(* CODESYS project Proje_1.project
   Title: Step
   Version: 0.0.0.0
   Author: MustafaZahid

Project tree, tasks and I/O mapping:
  MyController : TM241C24T/U, Schneider Electric, order no. TM241C24T/U, version 4.0.6.18
    application Application
      task MAST (cyclic, interval 20 ms, priority 15, watchdog 100 ms x 1) calls POU
      global variables GVL
      program POU [LD]
      FunctionBlocks/
        function block Motor_Administration [LD]
        function block Axis_Limits [LD]
    DI : Digital Inputs, Schneider Electric, version 4.0.6.18
        input  iwDI_IW0 : WORD  // IW0
        input  Application.POU.Sensor_1 : BOOL  // IW0.I0
        input  ibDI_IB1 : BYTE  // IB1
    DQ : Digital Outputs, Schneider Electric, version 4.0.6.18
        settings: Outputs Usage = 3
        output qwDQ_QW0 : WORD  // QW0
        output qbDQ_QB1 : BYTE  // QB1
    Counters : Counters, Schneider Electric, version 4.0.6.18
    Pulse_Generators : Pulse Generators, Schneider Electric, version 4.0.6.18
        settings: Instance name = 'Axis_1'; PROBE input History = 'old=0 new=-1'; REF input History = 'old=0 new=-1'; B output History = 'old=-1 new=1'; A output History = 'old=-1 new=0'; Temporary Instance name = 'Axis_1'
    Cartridge_1 : Cartridge, Schneider Electric, version 4.0.6.18
    IO_Bus : IO bus - TM3, Schneider Electric, version 4.0.6.18
    COM_Bus : COM bus, Schneider Electric, version 4.0.6.18
    Serial_Line_1 : Serial line, Schneider Electric, version 4.0.6.18
      SoMachine_Network_Manager : SoMachine-Network Manager, Schneider Electric, version 4.0.0.2
    Serial_Line_2 : Serial line, Schneider Electric, version 4.0.6.18
      Modbus_Manager : Modbus Manager, Schneider Electric, version 4.0.0.2
  text list GlobalTextList
*)

// MyController/Application/GVL
VAR_GLOBAL
END_VAR

// MyController/Application/POU
PROGRAM POU
VAR
	Motor_Administration_0: Motor_Administration;
	Power_En: BOOL;
	Reset_En: BOOL;
	Stop_En: BOOL;
	Set_Home: BOOL;
	MoveTo: BOOL;
	Return_Home: MC_MoveAbsolute_PTO;
	Return_En: BOOL;
	Axis_Limits_0: Axis_Limits;
	Set_Home_En: BOOL;
	PositiveMove_En: BOOL;
	NegativeMove_En: BOOL;
	BendingMachine: BOOL;
	Sensor_1: BOOL;
	Timer_1: TON;
	Timer_2: TON;
	Sensor_2: BOOL;
	Timer_3: TON;
	Timer_4: TON;
	Sensor_3: BOOL;
	Timer_5: TON;
	Timer_6: TON;
END_VAR

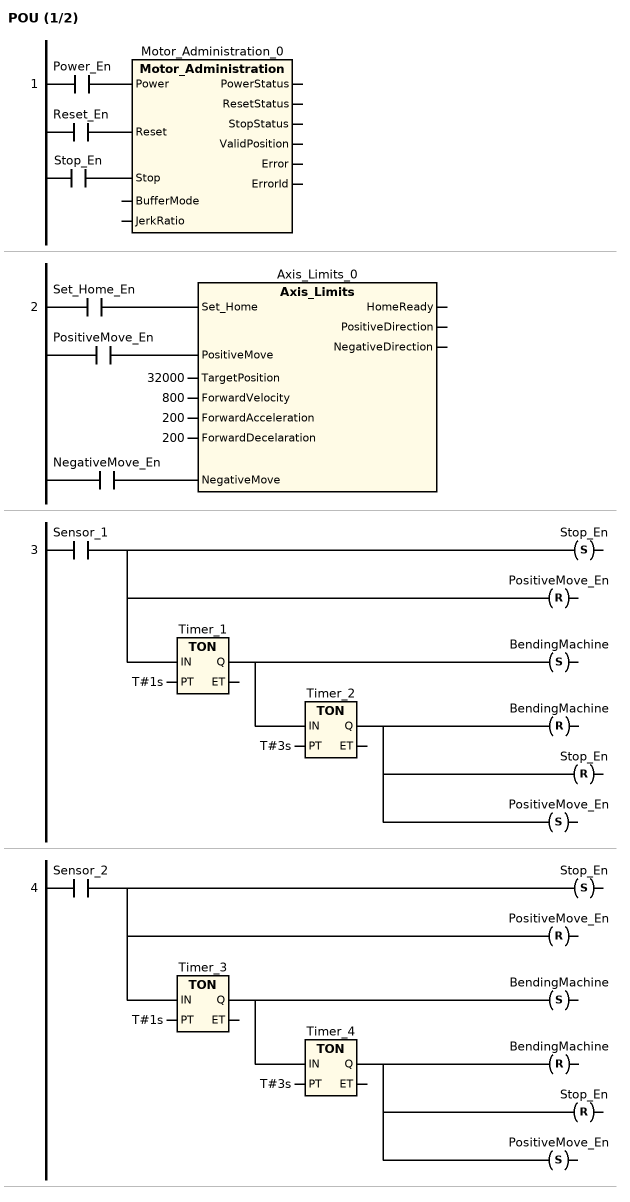
// NETWORK 1
Motor_Administration_0(Power := Power_En, Reset := Reset_En, Stop := Stop_En); // Motor_Administration

// NETWORK 2
Axis_Limits_0(
    Set_Home := Set_Home_En,
    PositiveMove := PositiveMove_En,
    TargetPosition := 32000,
    ForwardVelocity := 800,
    ForwardAcceleration := 200,
    ForwardDecelaration := 200,
    NegativeMove := NegativeMove_En); // Axis_Limits

// NETWORK 3
Stop_En S= Sensor_1;
PositiveMove_En R= Sensor_1;
Timer_1(IN := Sensor_1, PT := T#1s); // TON
BendingMachine S= Timer_1.Q;
Timer_2(IN := Timer_1.Q, PT := T#3s); // TON
BendingMachine R= Timer_2.Q;
Stop_En R= Timer_2.Q;
PositiveMove_En S= Timer_2.Q;

// NETWORK 4
Stop_En S= Sensor_2;
PositiveMove_En R= Sensor_2;
Timer_3(IN := Sensor_2, PT := T#1s); // TON
BendingMachine S= Timer_3.Q;
Timer_4(IN := Timer_3.Q, PT := T#3s); // TON
BendingMachine R= Timer_4.Q;
Stop_En R= Timer_4.Q;
PositiveMove_En S= Timer_4.Q;

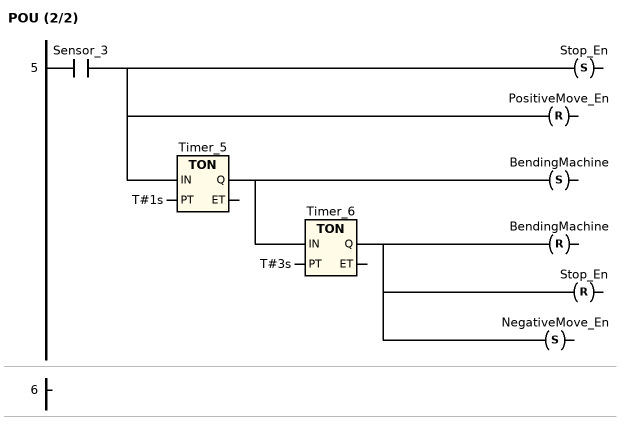
// NETWORK 5
Stop_En S= Sensor_3;
PositiveMove_En R= Sensor_3;
Timer_5(IN := Sensor_3, PT := T#1s); // TON
BendingMachine S= Timer_5.Q;
Timer_6(IN := Timer_5.Q, PT := T#3s); // TON
BendingMachine R= Timer_6.Q;
Stop_En R= Timer_6.Q;
NegativeMove_En S= Timer_6.Q;

// NETWORK 6

END_PROGRAM

// MyController/Application/FunctionBlocks/Motor_Administration
FUNCTION_BLOCK Motor_Administration
VAR_INPUT
	Power: BOOL;
	Reset: BOOL;
	Stop: BOOL;
	BufferMode: MC_BUFFER_MODE;
	JerkRatio: INT;
END_VAR
VAR_OUTPUT
	PowerStatus: BOOL;
	ResetStatus: BOOL;
	StopStatus: BOOL;
	ValidPosition: DINT;
	Error: BOOL;
	ErrorId: PTO_ERROR;
END_VAR
VAR
	MC_Power: MC_Power_PTO;
	MC_Reset: MC_Reset_PTO;
	MC_Stop: MC_Stop_PTO;
	MC_SetPosition: MC_SetPosition_PTO;
	MC_ReadActualPosition: MC_ReadActualPosition_PTO;
	MC_MoveAbsolute: MC_MoveAbsolute_PTO;
END_VAR

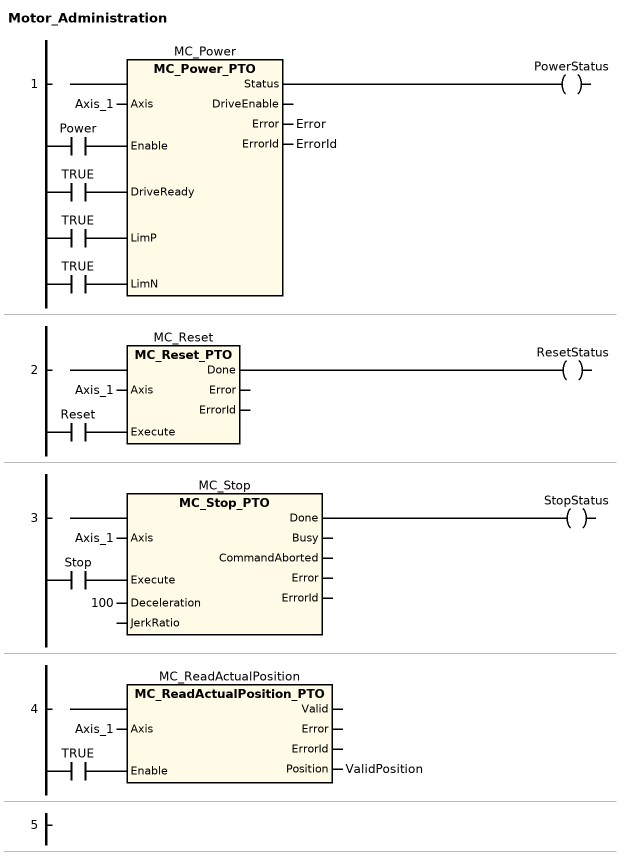
// NETWORK 1
MC_Power(
    Axis := Axis_1,
    Enable := Power,
    DriveReady := TRUE,
    LimP := TRUE,
    LimN := TRUE,
    Error => Error,
    ErrorId => ErrorId); // MC_Power_PTO
PowerStatus := MC_Power.Status;

// NETWORK 2
MC_Reset(Axis := Axis_1, Execute := Reset); // MC_Reset_PTO
ResetStatus := MC_Reset.Done;

// NETWORK 3
MC_Stop(Axis := Axis_1, Execute := Stop, Deceleration := 100); // MC_Stop_PTO
StopStatus := MC_Stop.Done;

// NETWORK 4
MC_ReadActualPosition(Axis := Axis_1, Enable := TRUE, Position => ValidPosition); // MC_ReadActualPosition_PTO

// NETWORK 5

END_FUNCTION_BLOCK

// MyController/Application/FunctionBlocks/Axis_Limits
FUNCTION_BLOCK Axis_Limits
VAR_INPUT
	Set_Home: BOOL;
	PositiveMove: BOOL;
	TargetPosition: DINT;
	ForwardVelocity: DINT;
	ForwardAcceleration: DINT;
	ForwardDecelaration: DINT;
	NegativeMove: BOOL;
END_VAR
VAR_OUTPUT
	HomeReady: BOOL;
	PositiveDirection: BOOL;
	NegativeDirection: BOOL;
END_VAR
VAR
	MC_Home: MC_Home_PTO;
	MC_Absolute_Positive: MC_MoveAbsolute_PTO;
	MC_Absolute_Negative: MC_MoveAbsolute_PTO;
END_VAR

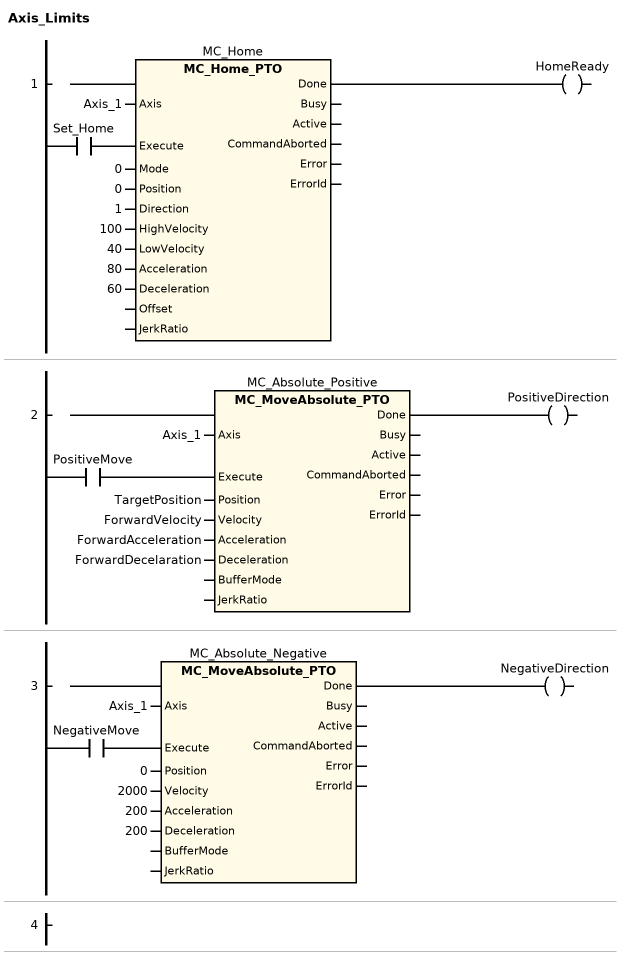
// NETWORK 1
MC_Home(
    Axis := Axis_1,
    Execute := Set_Home,
    Mode := 0,
    Position := 0,
    Direction := 1,
    HighVelocity := 100,
    LowVelocity := 40,
    Acceleration := 80,
    Deceleration := 60); // MC_Home_PTO
HomeReady := MC_Home.Done;

// NETWORK 2
MC_Absolute_Positive(
    Axis := Axis_1,
    Execute := PositiveMove,
    Position := TargetPosition,
    Velocity := ForwardVelocity,
    Acceleration := ForwardAcceleration,
    Deceleration := ForwardDecelaration); // MC_MoveAbsolute_PTO
PositiveDirection := MC_Absolute_Positive.Done;

// NETWORK 3
MC_Absolute_Negative(
    Axis := Axis_1,
    Execute := NegativeMove,
    Position := 0,
    Velocity := 2000,
    Acceleration := 200,
    Deceleration := 200); // MC_MoveAbsolute_PTO
NegativeDirection := MC_Absolute_Negative.Done;

// NETWORK 4

END_FUNCTION_BLOCK
